/// Enumeration of all possible component types
TYPE E_MachineArea :
(
	/// Common machine part
	eMachineArea_none := 0,
	eMachineArea_common,

	eMachineArea_max
);
END_TYPE

(* stored: Version 1.1.0.1, ProductVersion 3.1.4022.9
   DUT E_MachineArea: Id {1f82b0ad-04aa-4e81-b0b2-7db4e8b046a0} *)
